// TIA Portal V20 export
FUNCTION_BLOCK "CC_Station_Control"   // FB105, LAD
{ S7_Optimized_Access := 'TRUE' }
// stored: AutoNumber false, MemoryReserve 100, SetENOAutomatically false
   VAR_INPUT
      HMI_Reset : Bool;
      Station_Empty : Bool;
      Station_Occupied : Bool;
      Button_Seq_Forward : Bool;
      Button_Seq_Backward : Bool;
      HMI_Drive_Rollers_Down : Bool;
      HMI_Drive_Rollers_Up : Bool;
      HMI_Hydraulic_Down : Bool;
      HMI_Hydraulic_Up : Bool;
      HMI_Modules_Down : Bool;
      HMI_Modules_Up : Bool;
      HMI_Vibrating : Bool;
      CNT_DownPos1 : Bool;
      CNT_DownPos2 : Bool;
      CNT_UpPos1 : Bool;
      CNT_UpPos2 : Bool;
      Hydraulic_Roller_DownPos1 : Bool;
      Hydraulic_Roller_DownPos2 : Bool;
      Hydraulic_Roller_UpPos1 : Bool;
      Hydraulic_Roller_UpPos2 : Bool;
      Hydraulic_Unit_Ready : Bool;
      Drive_Roller_DownPos1 : Bool;
      Drive_Roller_DownPos2 : Bool;
      Drive_Roller_UpPos1 : Bool;
      Drive_Roller_UpPos2 : Bool;
      Modules_DownPos1 : Bool;
      Modules_DownPos2 : Bool;
      Modules_UpPos1 : Bool;
      Modules_UpPos2 : Bool;
   END_VAR
   VAR_OUTPUT
      Hydraulic_Unit : Bool;
      Hydraulic_Rollers_Up : Bool;
      Hydraulic_Rollers_Down : Bool;
      Vibration_Enable : Bool;
      Drive_Rollers_Up : Bool;
      Modules_Up : Bool;
   END_VAR
   VAR
      Hydraulic_Unit_Active : Bool;
      Hydraulic_Unit_TimerOff { S7_SetPoint := 'True'} : TON_TIME;
      Hydraulic_Unit_MC_Power { S7_SetPoint := 'True'} : MC_POWER;
      Hydraulic_Rollers { S7_SetPoint := 'True'} : "CC_Hydraulic_Rollers";
      Pneumatic_Rollers { S7_SetPoint := 'True'} : "CC_Pneumatic_Roller";
      Vibrator_Control { S7_SetPoint := 'True'} : "CC_Vibrator_Control";
      Sequence_Step { S7_SetPoint := 'True'} : Int;
      Req_Hydraulic_Rollers_Up : Bool;
      Req_Hydraulic_Rollers_Down : Bool;
      Req_Drive_Roller_Up : Bool;
      Req_Drive_Roller_Down : Bool;
      Req_Vibration_Enable : Bool;
      Req_Modules_Up : Bool;
      Req_Modules_Down : Bool;
      Sequence_Control { S7_SetPoint := 'True'} : "CC_Sequence_Control";
      Module_Control { S7_SetPoint := 'True'} : "CC_Vib_Modules";
      Hyd_Rollers_Up_whenMoving { S7_SetPoint := 'True'} : Bool;
   END_VAR
BEGIN

REGION Network 1: Centering devices position down
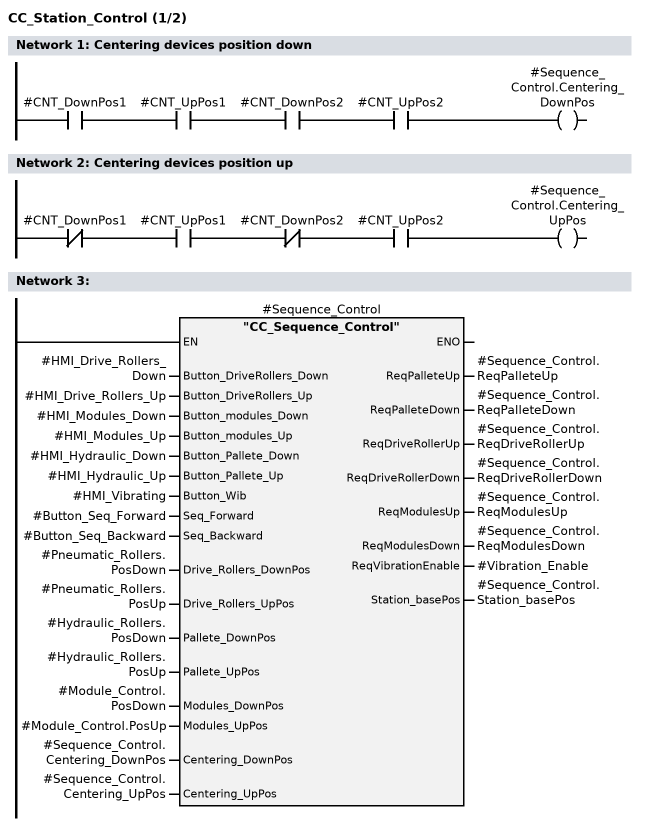
   RUNG wire#powerrail
      Contact( #CNT_DownPos1 )
      Contact( #CNT_UpPos1 )
      Contact( #CNT_DownPos2 )
      Contact( #CNT_UpPos2 )
      Coil( #Sequence_Control.Centering_DownPos )
   END_RUNG
   // the same network as SCL:
   #Sequence_Control.Centering_DownPos := #CNT_DownPos1 AND #CNT_UpPos1 AND #CNT_DownPos2 AND #CNT_UpPos2;
END_REGION

REGION Network 2: Centering devices position up
   RUNG wire#powerrail
      I_Contact( #CNT_DownPos1 )
      Contact( #CNT_UpPos1 )
      I_Contact( #CNT_DownPos2 )
      Contact( #CNT_UpPos2 )
      Coil( #Sequence_Control.Centering_UpPos )
   END_RUNG
   // the same network as SCL:
   #Sequence_Control.Centering_UpPos := NOT #CNT_DownPos1 AND #CNT_UpPos1 AND NOT #CNT_DownPos2 AND #CNT_UpPos2;
END_REGION

REGION Network 3
   RUNG wire#powerrail
      #Sequence_Control(Button_DriveRollers_Down := #HMI_Drive_Rollers_Down, Button_DriveRollers_Up := #HMI_Drive_Rollers_Up, Button_modules_Down := #HMI_Modules_Down, Button_modules_Up := #HMI_Modules_Up, Button_Pallete_Down := #HMI_Hydraulic_Down, Button_Pallete_Up := #HMI_Hydraulic_Up, Button_Wib := #HMI_Vibrating, Seq_Forward := #Button_Seq_Forward, Seq_Backward := #Button_Seq_Backward, Drive_Rollers_DownPos := #Pneumatic_Rollers.PosDown, Drive_Rollers_UpPos := #Pneumatic_Rollers.PosUp, Pallete_DownPos := #Hydraulic_Rollers.PosDown, Pallete_UpPos := #Hydraulic_Rollers.PosUp, Modules_DownPos := #Module_Control.PosDown, Modules_UpPos := #Module_Control.PosUp, Centering_DownPos := #Sequence_Control.Centering_DownPos, Centering_UpPos := #Sequence_Control.Centering_UpPos, ReqPalleteUp => #Sequence_Control.ReqPalleteUp, ReqPalleteDown => #Sequence_Control.ReqPalleteDown, ReqDriveRollerUp => #Sequence_Control.ReqDriveRollerUp, ReqDriveRollerDown => #Sequence_Control.ReqDriveRollerDown, ReqModulesUp => #Sequence_Control.ReqModulesUp, ReqModulesDown => #Sequence_Control.ReqModulesDown, ReqVibrationEnable => #Vibration_Enable, Station_basePos => #Sequence_Control.Station_basePos)
   END_RUNG
   // the same network as SCL:
   #Sequence_Control(Button_DriveRollers_Down := #HMI_Drive_Rollers_Down,   // "CC_Sequence_Control"
                     Button_DriveRollers_Up := #HMI_Drive_Rollers_Up,
                     Button_modules_Down := #HMI_Modules_Down,
                     Button_modules_Up := #HMI_Modules_Up,
                     Button_Pallete_Down := #HMI_Hydraulic_Down,
                     Button_Pallete_Up := #HMI_Hydraulic_Up,
                     Button_Wib := #HMI_Vibrating,
                     Seq_Forward := #Button_Seq_Forward,
                     Seq_Backward := #Button_Seq_Backward,
                     Drive_Rollers_DownPos := #Pneumatic_Rollers.PosDown,
                     Drive_Rollers_UpPos := #Pneumatic_Rollers.PosUp,
                     Pallete_DownPos := #Hydraulic_Rollers.PosDown,
                     Pallete_UpPos := #Hydraulic_Rollers.PosUp,
                     Modules_DownPos := #Module_Control.PosDown,
                     Modules_UpPos := #Module_Control.PosUp,
                     Centering_DownPos := #Sequence_Control.Centering_DownPos,
                     Centering_UpPos := #Sequence_Control.Centering_UpPos,
                     ReqPalleteUp => #Sequence_Control.ReqPalleteUp,
                     ReqPalleteDown => #Sequence_Control.ReqPalleteDown,
                     ReqDriveRollerUp => #Sequence_Control.ReqDriveRollerUp,
                     ReqDriveRollerDown => #Sequence_Control.ReqDriveRollerDown,
                     ReqModulesUp => #Sequence_Control.ReqModulesUp,
                     ReqModulesDown => #Sequence_Control.ReqModulesDown,
                     ReqVibrationEnable => #Vibration_Enable,
                     Station_basePos => #Sequence_Control.Station_basePos);
END_REGION

REGION Network 4: Hydraulic rollers control
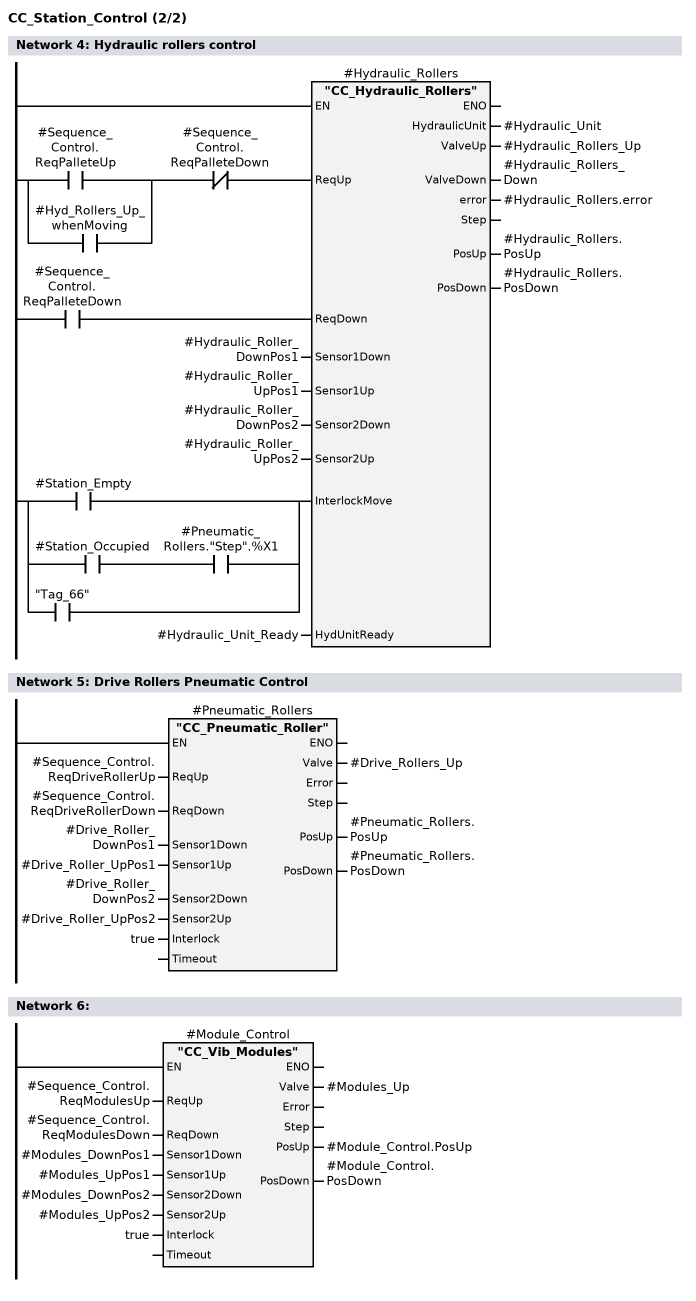
   RUNG wire#powerrail
      #Hydraulic_Rollers(ReqUp := wire#w2, ReqDown := wire#w3, InterlockMove := wire#w4, Sensor1Down := #Hydraulic_Roller_DownPos1, Sensor1Up := #Hydraulic_Roller_UpPos1, Sensor2Down := #Hydraulic_Roller_DownPos2, Sensor2Up := #Hydraulic_Roller_UpPos2, HydUnitReady := #Hydraulic_Unit_Ready, HydraulicUnit => #Hydraulic_Unit, ValveUp => #Hydraulic_Rollers_Up, ValveDown => #Hydraulic_Rollers_Down, error => #Hydraulic_Rollers.error, "Step" =>, PosUp => #Hydraulic_Rollers.PosUp, PosDown => #Hydraulic_Rollers.PosDown)
   END_RUNG
   RUNG wire#powerrail
      Contact( #Sequence_Control.ReqPalleteUp )
      wire#w1
      I_Contact( #Sequence_Control.ReqPalleteDown )
   END_RUNG wire#w2
   RUNG wire#powerrail
      Contact( #Hyd_Rollers_Up_whenMoving )
   END_RUNG wire#w1
   RUNG wire#powerrail
      Contact( #Sequence_Control.ReqPalleteDown )
   END_RUNG wire#w3
   RUNG wire#powerrail
      Contact( #Station_Empty )
   END_RUNG wire#w4
   RUNG wire#powerrail
      Contact( #Station_Occupied )
      Contact( #Pneumatic_Rollers."Step".%X1 )
   END_RUNG wire#w4
   RUNG wire#powerrail
      Contact( "Tag_66" )
   END_RUNG wire#w4
   // the same network as SCL:
   #Hydraulic_Rollers(ReqUp := (#Sequence_Control.ReqPalleteUp OR #Hyd_Rollers_Up_whenMoving) AND NOT #Sequence_Control.ReqPalleteDown,   // "CC_Hydraulic_Rollers"
                      ReqDown := #Sequence_Control.ReqPalleteDown,
                      Sensor1Down := #Hydraulic_Roller_DownPos1,
                      Sensor1Up := #Hydraulic_Roller_UpPos1,
                      Sensor2Down := #Hydraulic_Roller_DownPos2,
                      Sensor2Up := #Hydraulic_Roller_UpPos2,
                      InterlockMove := #Station_Empty OR (#Station_Occupied AND #Pneumatic_Rollers."Step".%X1) OR "Tag_66",
                      HydUnitReady := #Hydraulic_Unit_Ready,
                      HydraulicUnit => #Hydraulic_Unit,
                      ValveUp => #Hydraulic_Rollers_Up,
                      ValveDown => #Hydraulic_Rollers_Down,
                      error => #Hydraulic_Rollers.error,
                      PosUp => #Hydraulic_Rollers.PosUp,
                      PosDown => #Hydraulic_Rollers.PosDown);
END_REGION

REGION Network 5: Drive Rollers Pneumatic Control
   RUNG wire#powerrail
      #Pneumatic_Rollers(ReqUp := #Sequence_Control.ReqDriveRollerUp, ReqDown := #Sequence_Control.ReqDriveRollerDown, Sensor1Down := #Drive_Roller_DownPos1, Sensor1Up := #Drive_Roller_UpPos1, Sensor2Down := #Drive_Roller_DownPos2, Sensor2Up := #Drive_Roller_UpPos2, Interlock := true, Timeout :=, Valve => #Drive_Rollers_Up, Error =>, "Step" =>, PosUp => #Pneumatic_Rollers.PosUp, PosDown => #Pneumatic_Rollers.PosDown)
   END_RUNG
   // the same network as SCL:
   #Pneumatic_Rollers(ReqUp := #Sequence_Control.ReqDriveRollerUp,   // "CC_Pneumatic_Roller"
                      ReqDown := #Sequence_Control.ReqDriveRollerDown,
                      Sensor1Down := #Drive_Roller_DownPos1,
                      Sensor1Up := #Drive_Roller_UpPos1,
                      Sensor2Down := #Drive_Roller_DownPos2,
                      Sensor2Up := #Drive_Roller_UpPos2,
                      Interlock := true,
                      Valve => #Drive_Rollers_Up,
                      PosUp => #Pneumatic_Rollers.PosUp,
                      PosDown => #Pneumatic_Rollers.PosDown);
END_REGION

REGION Network 6
   RUNG wire#powerrail
      #Module_Control(ReqUp := #Sequence_Control.ReqModulesUp, ReqDown := #Sequence_Control.ReqModulesDown, Sensor1Down := #Modules_DownPos1, Sensor1Up := #Modules_UpPos1, Sensor2Down := #Modules_DownPos2, Sensor2Up := #Modules_UpPos2, Interlock := true, Timeout :=, Valve => #Modules_Up, Error =>, "Step" =>, PosUp => #Module_Control.PosUp, PosDown => #Module_Control.PosDown)
   END_RUNG
   // the same network as SCL:
   #Module_Control(ReqUp := #Sequence_Control.ReqModulesUp,   // "CC_Vib_Modules"
                   ReqDown := #Sequence_Control.ReqModulesDown,
                   Sensor1Down := #Modules_DownPos1,
                   Sensor1Up := #Modules_UpPos1,
                   Sensor2Down := #Modules_DownPos2,
                   Sensor2Up := #Modules_UpPos2,
                   Interlock := true,
                   Valve => #Modules_Up,
                   PosUp => #Module_Control.PosUp,
                   PosDown => #Module_Control.PosDown);
END_REGION
END_FUNCTION_BLOCK
